PROGRAM P_HeaterControl
VAR
	TempControl_1									: FB_Temp_Control;
	TempControl_2									: FB_Temp_Control;
	TempControl_3									: FB_Temp_Control;
	TempControl_4									: FB_Temp_Control;
	TempControl_5									: FB_Temp_Control;
	TempControl_6									: FB_Temp_Control;
END_VAR

// Calvin - P_HeaterControl
// Rev 1.00 - May 20, 2023

IF giActiveAlarm <> 1 AND tgb_HT_1_On THEN
	TempControl_1(
		Set_Point									:= tgr_HT_1_SP, 
		Temperature									:= tgr_TI_1, 
		I_Range 									:= tgr_HT_I_Range, 
		Pid_Cycle_Time								:= PID_CYCLE_TIME, 
		Pid_Kp										:= tgr_HT_P_Value, 
		Pid_Tn										:= tgr_HT_I_Value, 
		Pid_Tv										:= 0, 
		Pid_Td										:= 0,
		Base_Output									:= tgr_HT_1_Base_Output,
		Manual_Output								:= tgr_HT_1_Manual_Output,
		Output										=> HT_1_CTRL);
ELSE
	HT_1_CTRL										:= 0;
	HT_1_RELAY										:= FALSE;
END_IF
		
IF giActiveAlarm <> 1 AND tgb_HT_2_On THEN
	TempControl_2(
		Set_Point									:= tgr_HT_2_SP, 
		Temperature									:= tgr_TI_2, 
		I_Range 									:= tgr_HT_I_Range,
		Pid_Cycle_Time								:= PID_CYCLE_TIME, 
		Pid_Kp										:= tgr_HT_P_Value, 
		Pid_Tn										:= tgr_HT_I_Value, 
		Pid_Tv										:= 0, 
		Pid_Td										:= 0, 
		Base_Output									:= tgr_HT_2_Base_Output,
		Manual_Output								:= tgr_HT_2_Manual_Output, 
		Output										=> HT_2_CTRL);
ELSE
	HT_2_CTRL										:= 0;
	HT_2_RELAY										:= FALSE;
END_IF
		
IF giActiveAlarm <> 1 AND tgb_HT_3_On THEN
	TempControl_3(
		Set_Point									:= tgr_HT_3_SP, 
		Temperature									:= tgr_TI_3, 
		I_Range 									:= tgr_HT_I_Range,
		Pid_Cycle_Time								:= PID_CYCLE_TIME, 
		Pid_Kp										:= tgr_HT_P_Value, 
		Pid_Tn										:= tgr_HT_I_Value, 
		Pid_Tv										:= 0, 
		Pid_Td										:= 0, 
		Base_Output									:= tgr_HT_3_Base_Output,
		Manual_Output								:= tgr_HT_3_Manual_Output, 
		Output										=> HT_3_CTRL);
ELSE                                				
	HT_3_CTRL										:= 0;
	HT_3_RELAY										:= FALSE;
END_IF
		
IF giActiveAlarm <> 1 AND tgb_HT_4_On THEN
	TempControl_4(
		Set_Point									:= tgr_HT_4_SP, 
		Temperature									:= tgr_TI_4, 
		I_Range 									:= tgr_HT_I_Range,
		Pid_Cycle_Time								:= PID_CYCLE_TIME, 
		Pid_Kp										:= tgr_HT_P_Value, 
		Pid_Tn										:= tgr_HT_I_Value, 
		Pid_Tv										:= 0, 
		Pid_Td										:= 0,
		Base_Output									:= tgr_HT_4_Base_Output,
		Manual_Output								:= tgr_HT_4_Manual_Output, 
		Output										=> HT_4_CTRL);
ELSE                            				
	HT_4_CTRL										:= 0;
	HT_4_RELAY										:= FALSE;
END_IF                          	
		
IF giActiveAlarm <> 1 AND tgb_HT_5_On THEN
	TempControl_5(
		Set_Point									:= tgr_HT_5_SP, 
		Temperature									:= tgr_TI_5, 
		I_Range 									:= tgr_HT_I_Range,
		Pid_Cycle_Time								:= PID_CYCLE_TIME, 
		Pid_Kp										:= tgr_HT_P_Value, 
		Pid_Tn										:= tgr_HT_I_Value, 
		Pid_Tv										:= 0, 
		Pid_Td										:= 0,
		Base_Output									:= tgr_HT_5_Base_Output,
		Manual_Output								:= tgr_HT_5_Manual_Output,
		Output										=> HT_5_CTRL);
ELSE                        				
	HT_5_CTRL										:= 0;
	HT_5_RELAY										:= FALSE;
END_IF
		
IF giActiveAlarm <> 1 AND tgb_HT_6_On THEN
	TempControl_6(
		Set_Point									:= tgr_HT_6_SP, 
		Temperature									:= tgr_TI_6, 
		I_Range 									:= tgr_HT_I_Range,
		Pid_Cycle_Time								:= PID_CYCLE_TIME, 
		Pid_Kp										:= tgr_HT_P_Value, 
		Pid_Tn										:= tgr_HT_I_Value, 
		Pid_Tv										:= 0, 
		Pid_Td										:= 0, 
		Base_Output									:= tgr_HT_6_Base_Output,
		Manual_Output								:= tgr_HT_6_Manual_Output,
		Output										=> HT_6_CTRL);
ELSE                                	
	HT_6_CTRL							:= 0;
	HT_6_RELAY							:= FALSE;
END_IF                              	
	
tgr_HT_1_Ctrl						:= INT_TO_REAL(HT_1_CTRL);
tgr_HT_2_Ctrl						:= INT_TO_REAL(HT_2_CTRL);
tgr_HT_3_Ctrl						:= INT_TO_REAL(HT_3_CTRL);
tgr_HT_4_Ctrl						:= INT_TO_REAL(HT_4_CTRL);
tgr_HT_5_Ctrl						:= INT_TO_REAL(HT_5_CTRL);
tgr_HT_6_Ctrl						:= INT_TO_REAL(HT_6_CTRL);

END_PROGRAM

(* stored: Version 1.1.0.1, ProductVersion 3.1.4024.12
   POU P_HeaterControl: Id {031a7e95-28a9-4956-9d75-7514ddae1925}, SpecialFunc None *)
